{attribute 'linkalways'} 
{attribute 'no_explicit_call' := 'This FB is a CLASS and must be accessed using methods or properties'}
{attribute 'enable_dynamic_creation'}
FUNCTION_BLOCK ABSTRACT InterfaceDatatypeBase EXTENDS DatatypeBase IMPLEMENTS I_InterfaceDatatype
VAR
END_VAR

PROPERTY PUBLIC ABSTRACT Identifier : T_MAXSTRING
GET
END_GET
END_PROPERTY

PROPERTY PUBLIC IsUserDefined : BOOL
GET
IsUserDefined := FALSE;
END_GET
END_PROPERTY

METHOD PROTECTED OnSerializeTypeWith
VAR_INPUT
	Serializer : I_Serializer;
END_VAR
SUPER^.OnSerializeTypeWith(Serializer);
Serializer.AddKeyString('identifier',Identifier);
END_METHOD

METHOD PUBLIC TryCopyFrom : BOOL
VAR_INPUT
	Source : I_Datatype;
END_VAR
VAR
	sourceAsInterface : I_InterfaceDatatype;
END_VAR
IF NOT __QUERYINTERFACE(Source, sourceAsInterface) THEN
	RETURN;
END_IF

IF sourceAsInterface.Identifier <> Identifier THEN
	RETURN;
END_IF

TryCopyFrom := SUPER^.TryCopyFrom(Source);
END_METHOD

METHOD PUBLIC TryResolveAsInterfaceDatatype : BOOL
VAR_INPUT
	Destination : REFERENCE TO I_InterfaceDatatype;
END_VAR
Destination := THIS^;
TryResolveAsInterfaceDatatype := TRUE;
END_METHOD

PROPERTY PUBLIC TypeName : T_MAXSTRING
GET
TypeName := 'INTERFACE';
END_GET
END_PROPERTY

END_FUNCTION_BLOCK

(* stored: Version 1.1.0.1, ProductVersion 3.1.4024.12
   POU InterfaceDatatypeBase: Id {4cec4ea4-52ba-4a8f-9cb2-d853b09f5016}, SpecialFunc None
   Folder Protected: Id {33a6ae48-3763-4956-b972-7dd7c54cebcc}
   Property Identifier: Id {407a0089-b583-4518-bbe6-4cbec9996e45}
   Get Get: Id {320a3715-5f9c-42d8-8620-64702f1ff3ac}
   Property IsUserDefined: Id {d18b1469-03ed-4bc5-9302-58c4a2f1984c}
   Get Get: Id {edbfa430-1cb0-4dc2-8a1b-edf0ef849fd3}
   Method OnSerializeTypeWith: Id {5c4d3304-ef85-4e15-8f63-18c0ce3c1a59}
   Method TryCopyFrom: Id {0820a392-e788-497b-bba4-d8dc623c2d68}
   Method TryResolveAsInterfaceDatatype: Id {536062fb-ac06-4a91-9025-e106d39a9701}
   Property TypeName: Id {bab36bea-45e7-44e3-9000-b20c2aba1f60}
   Get Get: Id {b5598086-7a8f-4d1c-91d5-d64d64b933eb} *)
